INTERFACE I_MotionSystemApplication

METHOD Aborting : BOOL
VAR_INPUT
END_VAR
END_METHOD

METHOD Cycle : BOOL
VAR_INPUT
END_VAR
END_METHOD

METHOD Execute : UDINT
VAR_INPUT
END_VAR
END_METHOD

PROPERTY P_bMoverError : BOOL
GET
END_GET
SET
END_SET
END_PROPERTY

PROPERTY PUBLIC P_nAbortingSequence : UDINT
GET
END_GET
END_PROPERTY

PROPERTY PUBLIC P_nExecutingSequence : UDINT
GET
END_GET
END_PROPERTY

PROPERTY PUBLIC P_nResettingSequence : UDINT
GET
END_GET
END_PROPERTY

PROPERTY PUBLIC P_nStartingSequence : UDINT
GET
END_GET
END_PROPERTY

PROPERTY PUBLIC P_nStartupSequence : UDINT
GET
END_GET
END_PROPERTY

METHOD Resetting : BOOL
VAR_INPUT
END_VAR
END_METHOD

METHOD Starting : BOOL
VAR_INPUT
END_VAR
END_METHOD

METHOD Startup : BOOL
VAR_INPUT
END_VAR
END_METHOD

PROPERTY std : I_MotionSystem
GET
END_GET
SET
END_SET
END_PROPERTY

END_INTERFACE

(* stored: Version 1.1.0.1, ProductVersion 3.1.4024.9
   Itf I_MotionSystemApplication: Id {e7598d04-e0c3-40a6-86c8-2c0e70813362}
   Method Aborting: Id {6449c0d4-b573-4985-8f5f-5f5e3b093c91}
   Method Cycle: Id {da07f67e-baa2-495e-a207-1bf59d2fffb3}
   Method Execute: Id {f7fed176-5c6d-4de7-a24a-596d64fe196f}
   Property P_bMoverError: Id {09b76481-b8eb-4ed6-a9b0-f904e099bf33}
   Get Get: Id {8cc4a8b0-a9ef-4f67-8a56-ebaf2fce9538}
   Set Set: Id {d47b0568-3869-4d51-823b-e909b069ffc6}
   Property P_nAbortingSequence: Id {78b3c0c8-faf0-4d44-9658-651c8ace35aa}
   Get Get: Id {6760375f-ca2a-4030-8a5e-1ca0f5a3b2b9}
   Property P_nExecutingSequence: Id {ca9f24af-3daf-4ddb-b548-e483885c378b}
   Get Get: Id {3a450747-c5b1-4d88-ab14-924f6692492d}
   Property P_nResettingSequence: Id {bb318a4f-b92d-4c19-9572-d10640d2bb5a}
   Get Get: Id {7f67f8af-8b5f-41ad-b798-92ae01a0bdaa}
   Property P_nStartingSequence: Id {c7af3f23-c7bd-479c-b635-5c48cca21175}
   Get Get: Id {b7afb2e1-9612-40ed-b46c-ec465c7168ec}
   Property P_nStartupSequence: Id {e2ddb2af-0253-4c59-abd7-a95d56c766c2}
   Get Get: Id {cbc3d4d9-30fb-4263-b0de-b3f8a757cff7}
   Method Resetting: Id {43f0d798-b598-41ef-9716-ed187000313f}
   Method Starting: Id {a33ccdfa-d9f1-462f-87c0-020bbd11e729}
   Method Startup: Id {fcf88124-e8cc-40f7-a9b1-9e05853b68cd}
   Property std: Id {b102d276-a7e6-4eb9-8eae-922197c504af}
   Get Get: Id {052441c9-02cf-46f7-8b22-20ebc1c149c6}
   Set Set: Id {0f764bb4-31e2-4012-9455-e825e13d2944} *)
